DATA_BLOCK "KNX"
{ S7_Optimized_Access := 'FALSE' }
VERSION : 0.1
NON_RETAIN
   STRUCT
      DB_SIZE : Int;
      WO_DPT1 : "KNXDriver_GA";
      WO_DPT5 : "KNXDriver_GA";
      WO_DPT9 : "KNXDriver_GA";
      RO_DPT9 : "KNXDriver_GA";
      WO_DPT14 : "KNXDriver_GA";
      RO_DPT14 : "KNXDriver_GA";
      WO_DPT233 : "KNXDriver_GA_232";
      RO_DPT232 : "KNXDriver_GA_232";
   END_STRUCT;


BEGIN
   WO_DPT1.GA := 0001008;
   WO_DPT1."Type" := 1;
   WO_DPT1.WRITE_ONLY := true;
   WO_DPT1.val_real := 120.0;
   WO_DPT5.GA := 0001000;
   WO_DPT5."Type" := 5;
   WO_DPT5.WRITE_ONLY := true;
   WO_DPT9.GA := 0001008;
   WO_DPT9."Type" := 9;
   WO_DPT9.WRITE_ONLY := true;
   RO_DPT9.GA := 0001008;
   RO_DPT9."Type" := 9;
   RO_DPT9."READ_ONLY" := true;
   WO_DPT14."Type" := 14;
   WO_DPT14.WRITE_ONLY := true;
   RO_DPT14.GA := 0001230;
   RO_DPT14."Type" := 14;
   RO_DPT14."READ_ONLY" := true;
   WO_DPT233.GA := 0001232;
   WO_DPT233."Type" := 232;
   WO_DPT233.WRITE_ONLY := true;
   RO_DPT232.GA := 0001233;
   RO_DPT232."Type" := 232;
   RO_DPT232."READ_ONLY" := true;
   RO_DPT232.WRITE_ONLY := false;

END_DATA_BLOCK

